// TIA Portal project "hw2.1" (V15.1)

(* hardware
DEVICE "S7-1200 station_1"  S7-1200 Station
   slot 0: "Rack_0"  S7-1200 Rack  Rack  V1.0
   slot 1: "PLC_1"  CPU 1214C DC/DC/DC  6ES7 214-1AG40-0XB0  V4.2
*)

// ===== PLC "PLC_1"  CPU 1214C DC/DC/DC =====

VAR_GLOBAL   // PLC tag table "Default tag table"
   "sistem" AT %Q0.0 : Bool;
   "stop" AT %I0.0 : Bool;
   "X0_sensor" AT %I0.1 : Bool;
   "Y0_open_door" AT %Q0.1 : Bool;
   "X2_limit" AT %I0.2 : Bool;
   "bekleme" AT %Q0.2 : Bool;
   "X1_limit" AT %I0.3 : Bool;
   "Y1" AT %Q0.3 : Bool;
END_VAR

// folder: System blocks/Program resources

DATA_BLOCK "IEC_Timer_0_DB_1"   // DB2
{ S7_Optimized_Access := 'TRUE' }
AUTHOR : Simatic
FAMILY : IEC
NAME : IEC_TMR
VERSION : 1.0
// stored: InstanceOfName IEC_TIMER
"IEC_TIMER"
BEGIN
END_DATA_BLOCK

// folder: (top level)

ORGANIZATION_BLOCK "Main"   // OB1, LAD, ProgramCycle
TITLE = "Main Program Sweep (Cycle)"
{ S7_Optimized_Access := 'TRUE' }
VERSION : 0.1
   VAR_INPUT
      Initial_Call : Bool;   // Initial call of this OB
      Remanence : Bool;   // =True, if remanent data are available
   END_VAR
BEGIN

REGION Network 1
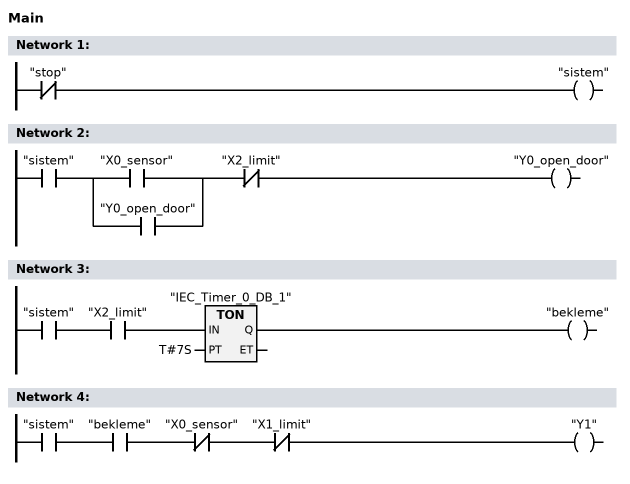
   RUNG wire#powerrail
      I_Contact( "stop" )
      Coil( "sistem" )
   END_RUNG
   // the same network as SCL:
   "sistem" := NOT "stop";
END_REGION

REGION Network 2
   RUNG wire#powerrail
      Contact( "sistem" )
      wire#w1
      Contact( "X0_sensor" )
      wire#w2
      I_Contact( "X2_limit" )
      Coil( "Y0_open_door" )
   END_RUNG
   RUNG wire#w1
      Contact( "Y0_open_door" )
   END_RUNG wire#w2
   // the same network as SCL:
   "Y0_open_door" := "sistem" AND ("X0_sensor" OR "Y0_open_door") AND NOT "X2_limit";
END_REGION

REGION Network 3
   "IEC_Timer_0_DB_1".TON(IN := "sistem" AND "X2_limit", PT := T#7S);
   "bekleme" := "IEC_Timer_0_DB_1".Q;
END_REGION

REGION Network 4
   RUNG wire#powerrail
      Contact( "sistem" )
      Contact( "bekleme" )
      I_Contact( "X0_sensor" )
      I_Contact( "X1_limit" )
      Coil( "Y1" )
   END_RUNG
   // the same network as SCL:
   "Y1" := "sistem" AND "bekleme" AND NOT "X0_sensor" AND NOT "X1_limit";
END_REGION
END_ORGANIZATION_BLOCK